% RSLogix 500 project 07_P10_ASHLEY_J.RSS, saved by version 8.30.00.16 %
PROJECT "UNTITLED"    % processor: Bul.1763 MicroLogix 1100 Series B %

PROGRAM FILES
  LAD 2 "MAIN"  5 rungs
  LAD 3 "IO"  8 rungs
  LAD 4 "HOA_CTRLS"  10 rungs
  LAD 5 "CONTROLS"  7 rungs
  LAD 6 "ALARMS"  14 rungs

DATA FILES
  O0 OUTPUT  4 elements
  I1 INPUT  6 elements
  S2 STATUS  66 elements
  B3 BINARY  10 elements
  T4 TIMER  4 elements
  C5 COUNTER  1 elements
  R6 CONTROL  1 elements
  N7 INTEGER  4 elements
  F8 FLOAT  1 elements

LADDER 2 "MAIN"
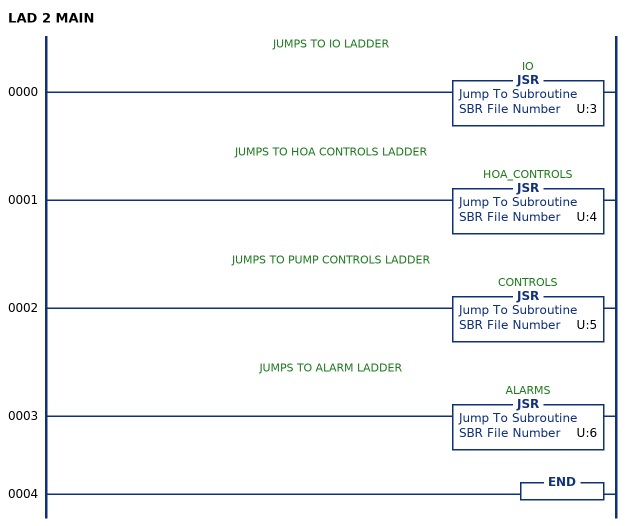
% Rung: 0 %
% JUMPS TO IO LADDER %
SOR JSR U:3 EOR
%   U:3  "IO" %
% Rung: 1 %
% JUMPS TO HOA CONTROLS LADDER %
SOR JSR U:4 EOR
%   U:4  "HOA_CONTROLS" %
% Rung: 2 %
% JUMPS TO PUMP CONTROLS LADDER %
SOR JSR U:5 EOR
%   U:5  "CONTROLS" %
% Rung: 3 %
% JUMPS TO ALARM LADDER %
SOR JSR U:6 EOR
%   U:6  "ALARMS" %
% Rung: 4 %
SOR END EOR

LADDER 3 "IO"
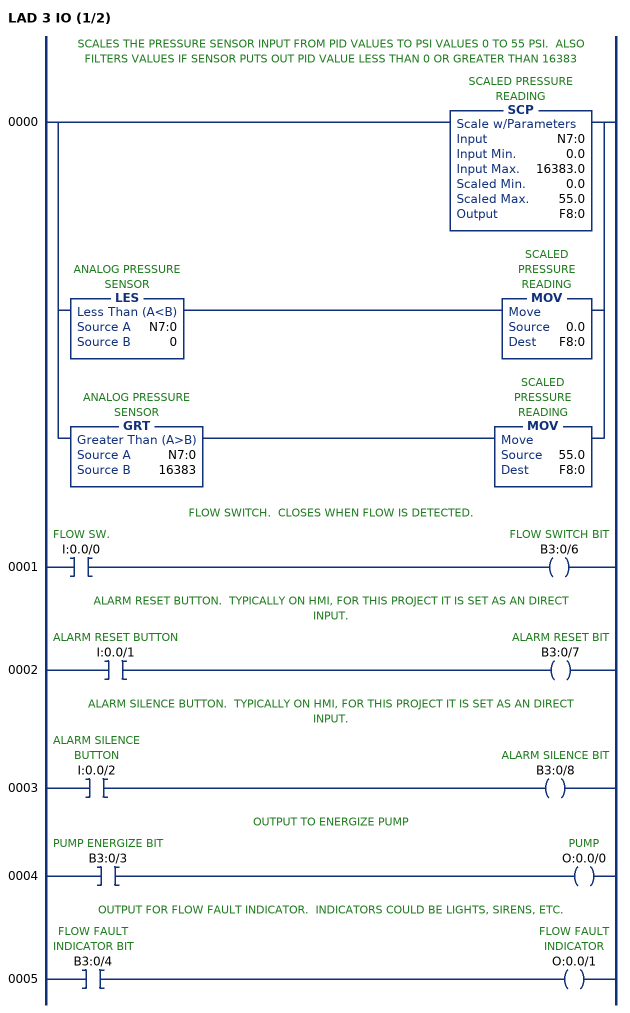
% Rung: 0 %
% SCALES THE PRESSURE SENSOR INPUT FROM PID VALUES TO PSI VALUES 0 TO 55 PSI.  ALSO FILTERS VALUES IF SENSOR PUTS OUT PID VALUE LESS THAN 0 OR GREATER THAN 16383 %
SOR BST SCP N7:0 0.0 16383.0 0.0 55.0 F8:0 NXB LES N7:0 0 MOV 0.0 F8:0 NXB GRT N7:0 16383 MOV 55.0 F8:0 BND EOR
%   N7:0  "ANALOG PRESSURE SENSOR" %
%   F8:0  "SCALED PRESSURE READING" %
% Rung: 1 %
% FLOW SWITCH.  CLOSES WHEN FLOW IS DETECTED. %
SOR XIC I:0.0/0 OTE B3:0/6 EOR
%   I:0.0/0  "FLOW SW." %
%   B3:0/6  "FLOW SWITCH BIT" %
% Rung: 2 %
% ALARM RESET BUTTON.  TYPICALLY ON HMI, FOR THIS PROJECT IT IS SET AS AN DIRECT INPUT. %
SOR XIC I:0.0/1 OTE B3:0/7 EOR
%   I:0.0/1  "ALARM RESET BUTTON" %
%   B3:0/7  "ALARM RESET BIT" %
% Rung: 3 %
% ALARM SILENCE BUTTON.  TYPICALLY ON HMI, FOR THIS PROJECT IT IS SET AS AN DIRECT INPUT. %
SOR XIC I:0.0/2 OTE B3:0/8 EOR
%   I:0.0/2  "ALARM SILENCE BUTTON" %
%   B3:0/8  "ALARM SILENCE BIT" %
% Rung: 4 %
% OUTPUT TO ENERGIZE PUMP %
SOR XIC B3:0/3 OTE O:0.0/0 EOR
%   B3:0/3  "PUMP ENERGIZE BIT" %
%   O:0.0/0  "PUMP" %
% Rung: 5 %
% OUTPUT FOR FLOW FAULT INDICATOR.  INDICATORS COULD BE LIGHTS, SIRENS, ETC. %
SOR XIC B3:0/4 OTE O:0.0/1 EOR
%   B3:0/4  "FLOW FAULT INDICATOR BIT" %
%   O:0.0/1  "FLOW FAULT INDICATOR" %

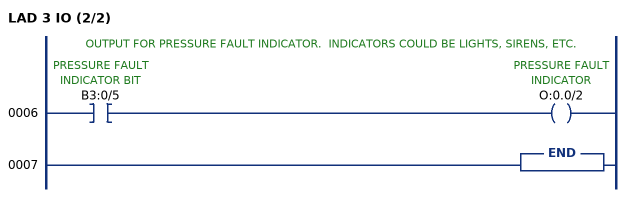
% Rung: 6 %
% OUTPUT FOR PRESSURE FAULT INDICATOR.  INDICATORS COULD BE LIGHTS, SIRENS, ETC. %
SOR XIC B3:0/5 OTE O:0.0/2 EOR
%   B3:0/5  "PRESSURE FAULT INDICATOR BIT" %
%   O:0.0/2  "PRESSURE FAULT INDICATOR" %
% Rung: 7 %
SOR END EOR

LADDER 4 "HOA_CTRLS"
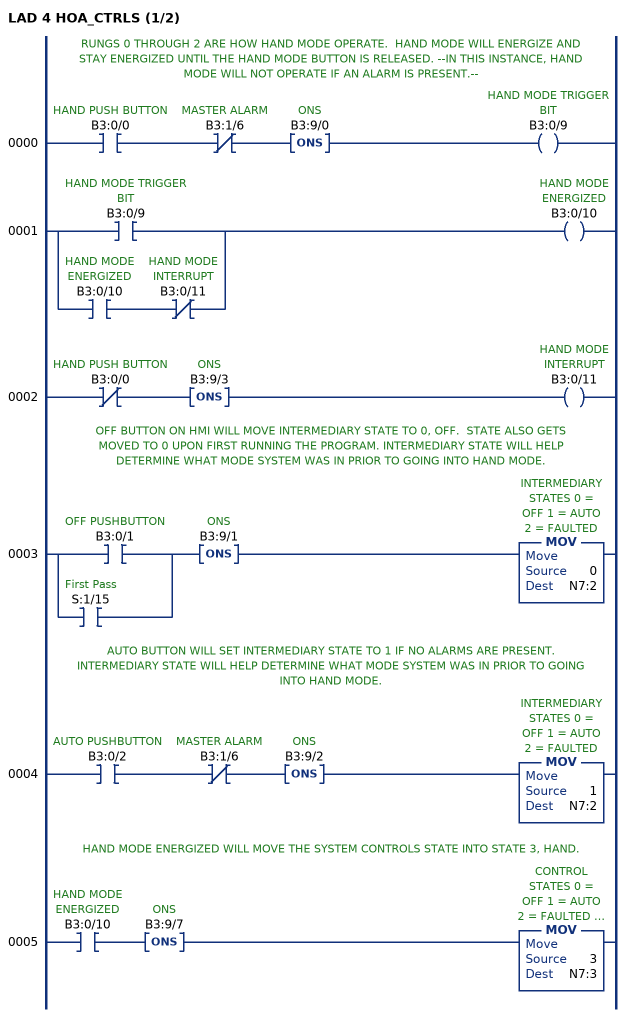
% Rung: 0 %
% RUNGS 0 THROUGH 2 ARE HOW HAND MODE OPERATE.  HAND MODE WILL ENERGIZE AND STAY ENERGIZED UNTIL THE HAND MODE BUTTON IS RELEASED. --IN THIS INSTANCE, HAND MODE WILL NOT OPERATE IF AN ALARM IS PRESENT.-- %
SOR XIC B3:0/0 XIO B3:1/6 ONS B3:9/0 OTE B3:0/9 EOR
%   B3:0/0  "HAND PUSH BUTTON" %
%   B3:1/6  "MASTER ALARM" %
%   B3:9/0  "ONS" %
%   B3:0/9  "HAND MODE TRIGGER BIT" %
% Rung: 1 %
SOR BST XIC B3:0/9 NXB XIC B3:0/10 XIO B3:0/11 BND OTE B3:0/10 EOR
%   B3:0/9  "HAND MODE TRIGGER BIT" %
%   B3:0/10  "HAND MODE ENERGIZED" %
%   B3:0/11  "HAND MODE INTERRUPT" %
% Rung: 2 %
SOR XIO B3:0/0 ONS B3:9/3 OTE B3:0/11 EOR
%   B3:0/0  "HAND PUSH BUTTON" %
%   B3:9/3  "ONS" %
%   B3:0/11  "HAND MODE INTERRUPT" %
% Rung: 3 %
% OFF BUTTON ON HMI WILL MOVE INTERMEDIARY STATE TO 0, OFF.  STATE ALSO GETS MOVED TO 0 UPON FIRST RUNNING THE PROGRAM. INTERMEDIARY STATE WILL HELP DETERMINE WHAT MODE SYSTEM WAS IN PRIOR TO GOING INTO HAND MODE. %
SOR BST XIC B3:0/1 NXB XIC S:1/15 BND ONS B3:9/1 MOV 0 N7:2 EOR
%   B3:0/1  "OFF PUSHBUTTON" %
%   S:1/15  "First Pass" %
%   B3:9/1  "ONS" %
%   N7:2  "INTERMEDIARY STATES 0 = OFF 1 = AUTO 2 = FAULTED" %
% Rung: 4 %
% AUTO BUTTON WILL SET INTERMEDIARY STATE TO 1 IF NO ALARMS ARE PRESENT.  INTERMEDIARY STATE WILL HELP DETERMINE WHAT MODE SYSTEM WAS IN PRIOR TO GOING INTO HAND MODE. %
SOR XIC B3:0/2 XIO B3:1/6 ONS B3:9/2 MOV 1 N7:2 EOR
%   B3:0/2  "AUTO PUSHBUTTON" %
%   B3:1/6  "MASTER ALARM" %
%   B3:9/2  "ONS" %
%   N7:2  "INTERMEDIARY STATES 0 = OFF 1 = AUTO 2 = FAULTED" %
% Rung: 5 %
% HAND MODE ENERGIZED WILL MOVE THE SYSTEM CONTROLS STATE INTO STATE 3, HAND. %
SOR XIC B3:0/10 ONS B3:9/7 MOV 3 N7:3 EOR
%   B3:0/10  "HAND MODE ENERGIZED" %
%   B3:9/7  "ONS" %
%   N7:3  "CONTROL STATES 0 = OFF 1 = AUTO 2 = FAULTED 3 = HAND" %

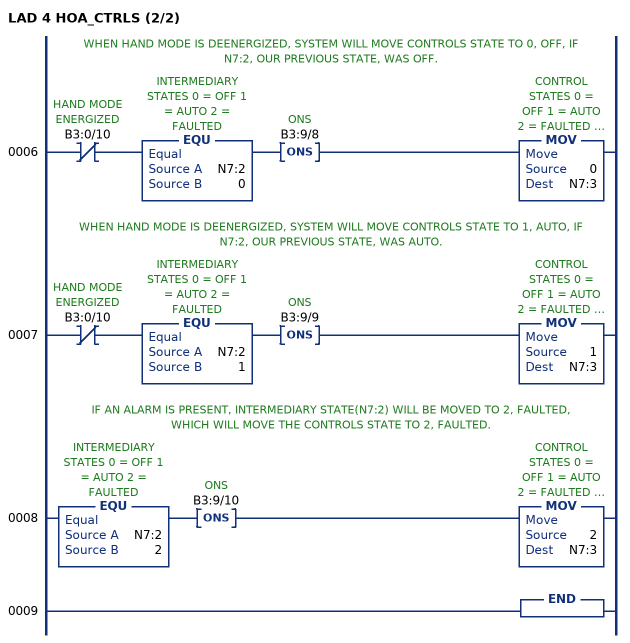
% Rung: 6 %
% WHEN HAND MODE IS DEENERGIZED, SYSTEM WILL MOVE CONTROLS STATE TO 0, OFF, IF N7:2, OUR PREVIOUS STATE, WAS OFF. %
SOR XIO B3:0/10 EQU N7:2 0 ONS B3:9/8 MOV 0 N7:3 EOR
%   B3:0/10  "HAND MODE ENERGIZED" %
%   N7:2  "INTERMEDIARY STATES 0 = OFF 1 = AUTO 2 = FAULTED" %
%   B3:9/8  "ONS" %
%   N7:3  "CONTROL STATES 0 = OFF 1 = AUTO 2 = FAULTED 3 = HAND" %
% Rung: 7 %
% WHEN HAND MODE IS DEENERGIZED, SYSTEM WILL MOVE CONTROLS STATE TO 1, AUTO, IF N7:2, OUR PREVIOUS STATE, WAS AUTO. %
SOR XIO B3:0/10 EQU N7:2 1 ONS B3:9/9 MOV 1 N7:3 EOR
%   B3:0/10  "HAND MODE ENERGIZED" %
%   N7:2  "INTERMEDIARY STATES 0 = OFF 1 = AUTO 2 = FAULTED" %
%   B3:9/9  "ONS" %
%   N7:3  "CONTROL STATES 0 = OFF 1 = AUTO 2 = FAULTED 3 = HAND" %
% Rung: 8 %
% IF AN ALARM IS PRESENT, INTERMEDIARY STATE(N7:2) WILL BE MOVED TO 2, FAULTED, WHICH WILL MOVE THE CONTROLS STATE TO 2, FAULTED. %
SOR EQU N7:2 2 ONS B3:9/10 MOV 2 N7:3 EOR
%   N7:2  "INTERMEDIARY STATES 0 = OFF 1 = AUTO 2 = FAULTED" %
%   B3:9/10  "ONS" %
%   N7:3  "CONTROL STATES 0 = OFF 1 = AUTO 2 = FAULTED 3 = HAND" %
% Rung: 9 %
SOR END EOR

LADDER 5 "CONTROLS"
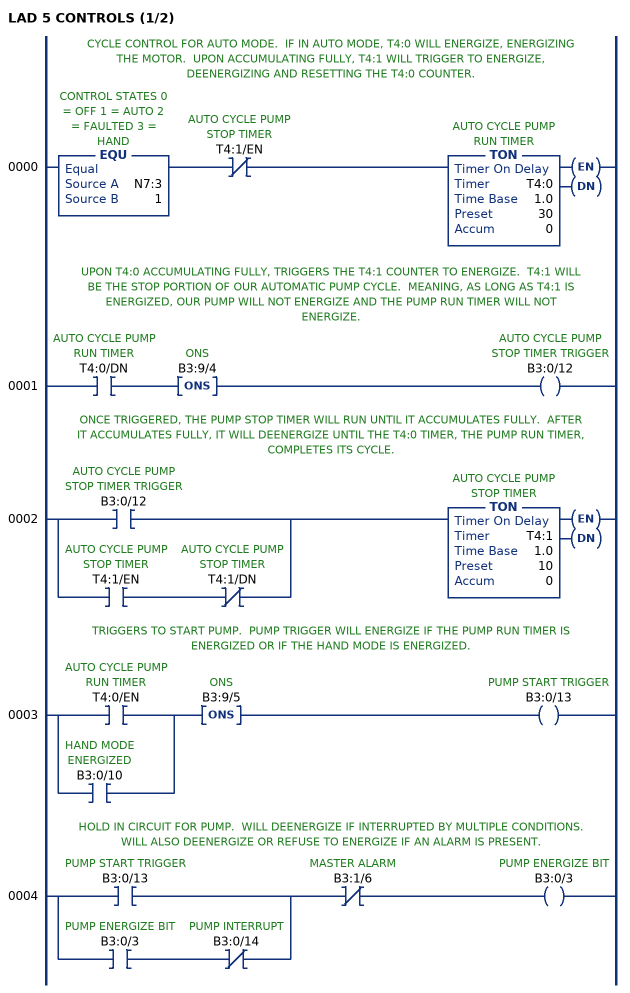
% Rung: 0 %
% CYCLE CONTROL FOR AUTO MODE.  IF IN AUTO MODE, T4:0 WILL ENERGIZE, ENERGIZING THE MOTOR.  UPON ACCUMULATING FULLY, T4:1 WILL TRIGGER TO ENERGIZE, DEENERGIZING AND RESETTING THE T4:0 COUNTER. %
SOR EQU N7:3 1 XIO T4:1/EN TON T4:0 1.0 30 0 EOR
%   N7:3  "CONTROL STATES 0 = OFF 1 = AUTO 2 = FAULTED 3 = HAND" %
%   T4:1  "AUTO CYCLE PUMP STOP TIMER" %
%   T4:0  "AUTO CYCLE PUMP RUN TIMER" %
% Rung: 1 %
% UPON T4:0 ACCUMULATING FULLY, TRIGGERS THE T4:1 COUNTER TO ENERGIZE.  T4:1 WILL BE THE STOP PORTION OF OUR AUTOMATIC PUMP CYCLE.  MEANING, AS LONG AS T4:1 IS ENERGIZED, OUR PUMP WILL NOT ENERGIZE AND THE PUMP RUN TIMER WILL NOT ENERGIZE. %
SOR XIC T4:0/DN ONS B3:9/4 OTE B3:0/12 EOR
%   T4:0  "AUTO CYCLE PUMP RUN TIMER" %
%   B3:9/4  "ONS" %
%   B3:0/12  "AUTO CYCLE PUMP STOP TIMER TRIGGER" %
% Rung: 2 %
% ONCE TRIGGERED, THE PUMP STOP TIMER WILL RUN UNTIL IT ACCUMULATES FULLY.  AFTER IT ACCUMULATES FULLY, IT WILL DEENERGIZE UNTIL THE T4:0 TIMER, THE PUMP RUN TIMER, COMPLETES ITS CYCLE. %
SOR BST XIC B3:0/12 NXB XIC T4:1/EN XIO T4:1/DN BND TON T4:1 1.0 10 0 EOR
%   B3:0/12  "AUTO CYCLE PUMP STOP TIMER TRIGGER" %
%   T4:1  "AUTO CYCLE PUMP STOP TIMER" %
% Rung: 3 %
% TRIGGERS TO START PUMP.  PUMP TRIGGER WILL ENERGIZE IF THE PUMP RUN TIMER IS ENERGIZED OR IF THE HAND MODE IS ENERGIZED. %
SOR BST XIC T4:0/EN NXB XIC B3:0/10 BND ONS B3:9/5 OTE B3:0/13 EOR
%   T4:0  "AUTO CYCLE PUMP RUN TIMER" %
%   B3:0/10  "HAND MODE ENERGIZED" %
%   B3:9/5  "ONS" %
%   B3:0/13  "PUMP START TRIGGER" %
% Rung: 4 %
% HOLD IN CIRCUIT FOR PUMP.  WILL DEENERGIZE IF INTERRUPTED BY MULTIPLE CONDITIONS.  WILL ALSO DEENERGIZE OR REFUSE TO ENERGIZE IF AN ALARM IS PRESENT. %
SOR BST XIC B3:0/13 NXB XIC B3:0/3 XIO B3:0/14 BND XIO B3:1/6 OTE B3:0/3 EOR
%   B3:0/13  "PUMP START TRIGGER" %
%   B3:0/3  "PUMP ENERGIZE BIT" %
%   B3:0/14  "PUMP INTERRUPT" %
%   B3:1/6  "MASTER ALARM" %

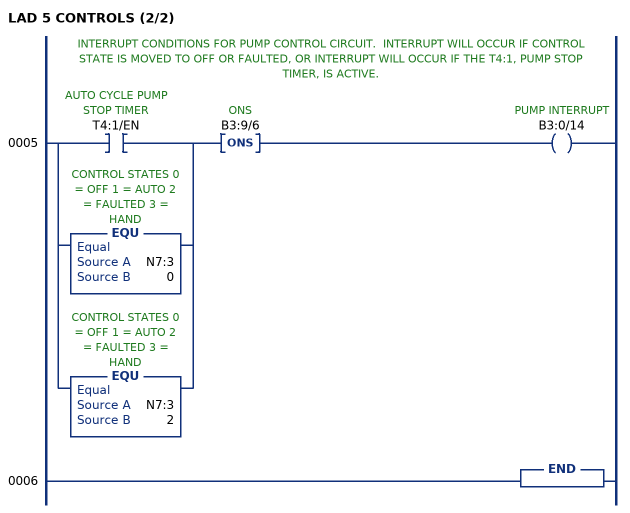
% Rung: 5 %
% INTERRUPT CONDITIONS FOR PUMP CONTROL CIRCUIT.  INTERRUPT WILL OCCUR IF CONTROL STATE IS MOVED TO OFF OR FAULTED, OR INTERRUPT WILL OCCUR IF THE T4:1, PUMP STOP TIMER, IS ACTIVE. %
SOR BST XIC T4:1/EN NXB EQU N7:3 0 NXB EQU N7:3 2 BND ONS B3:9/6 OTE B3:0/14 EOR
%   T4:1  "AUTO CYCLE PUMP STOP TIMER" %
%   N7:3  "CONTROL STATES 0 = OFF 1 = AUTO 2 = FAULTED 3 = HAND" %
%   B3:9/6  "ONS" %
%   B3:0/14  "PUMP INTERRUPT" %
% Rung: 6 %
SOR END EOR

LADDER 6 "ALARMS"
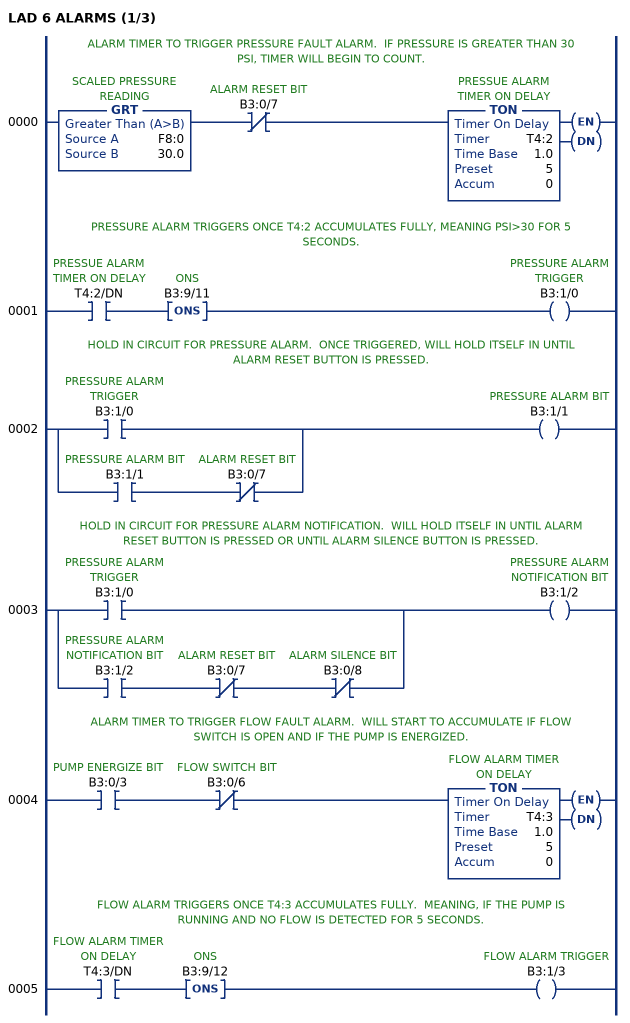
% Rung: 0 %
% ALARM TIMER TO TRIGGER PRESSURE FAULT ALARM.  IF PRESSURE IS GREATER THAN 30 PSI, TIMER WILL BEGIN TO COUNT. %
SOR GRT F8:0 30.0 XIO B3:0/7 TON T4:2 1.0 5 0 EOR
%   F8:0  "SCALED PRESSURE READING" %
%   B3:0/7  "ALARM RESET BIT" %
%   T4:2  "PRESSUE ALARM TIMER ON DELAY" %
% Rung: 1 %
% PRESSURE ALARM TRIGGERS ONCE T4:2 ACCUMULATES FULLY, MEANING PSI>30 FOR 5 SECONDS. %
SOR XIC T4:2/DN ONS B3:9/11 OTE B3:1/0 EOR
%   T4:2  "PRESSUE ALARM TIMER ON DELAY" %
%   B3:9/11  "ONS" %
%   B3:1/0  "PRESSURE ALARM TRIGGER" %
% Rung: 2 %
% HOLD IN CIRCUIT FOR PRESSURE ALARM.  ONCE TRIGGERED, WILL HOLD ITSELF IN UNTIL ALARM RESET BUTTON IS PRESSED. %
SOR BST XIC B3:1/0 NXB XIC B3:1/1 XIO B3:0/7 BND OTE B3:1/1 EOR
%   B3:1/0  "PRESSURE ALARM TRIGGER" %
%   B3:1/1  "PRESSURE ALARM BIT" %
%   B3:0/7  "ALARM RESET BIT" %
% Rung: 3 %
% HOLD IN CIRCUIT FOR PRESSURE ALARM NOTIFICATION.  WILL HOLD ITSELF IN UNTIL ALARM RESET BUTTON IS PRESSED OR UNTIL ALARM SILENCE BUTTON IS PRESSED. %
SOR BST XIC B3:1/0 NXB XIC B3:1/2 XIO B3:0/7 XIO B3:0/8 BND OTE B3:1/2 EOR
%   B3:1/0  "PRESSURE ALARM TRIGGER" %
%   B3:1/2  "PRESSURE ALARM NOTIFICATION BIT" %
%   B3:0/7  "ALARM RESET BIT" %
%   B3:0/8  "ALARM SILENCE BIT" %
% Rung: 4 %
% ALARM TIMER TO TRIGGER FLOW FAULT ALARM.  WILL START TO ACCUMULATE IF FLOW SWITCH IS OPEN AND IF THE PUMP IS ENERGIZED. %
SOR XIC B3:0/3 XIO B3:0/6 TON T4:3 1.0 5 0 EOR
%   B3:0/3  "PUMP ENERGIZE BIT" %
%   B3:0/6  "FLOW SWITCH BIT" %
%   T4:3  "FLOW ALARM TIMER ON DELAY" %
% Rung: 5 %
% FLOW ALARM TRIGGERS ONCE T4:3 ACCUMULATES FULLY.  MEANING, IF THE PUMP IS RUNNING AND NO FLOW IS DETECTED FOR 5 SECONDS. %
SOR XIC T4:3/DN ONS B3:9/12 OTE B3:1/3 EOR
%   T4:3  "FLOW ALARM TIMER ON DELAY" %
%   B3:9/12  "ONS" %
%   B3:1/3  "FLOW ALARM TRIGGER" %

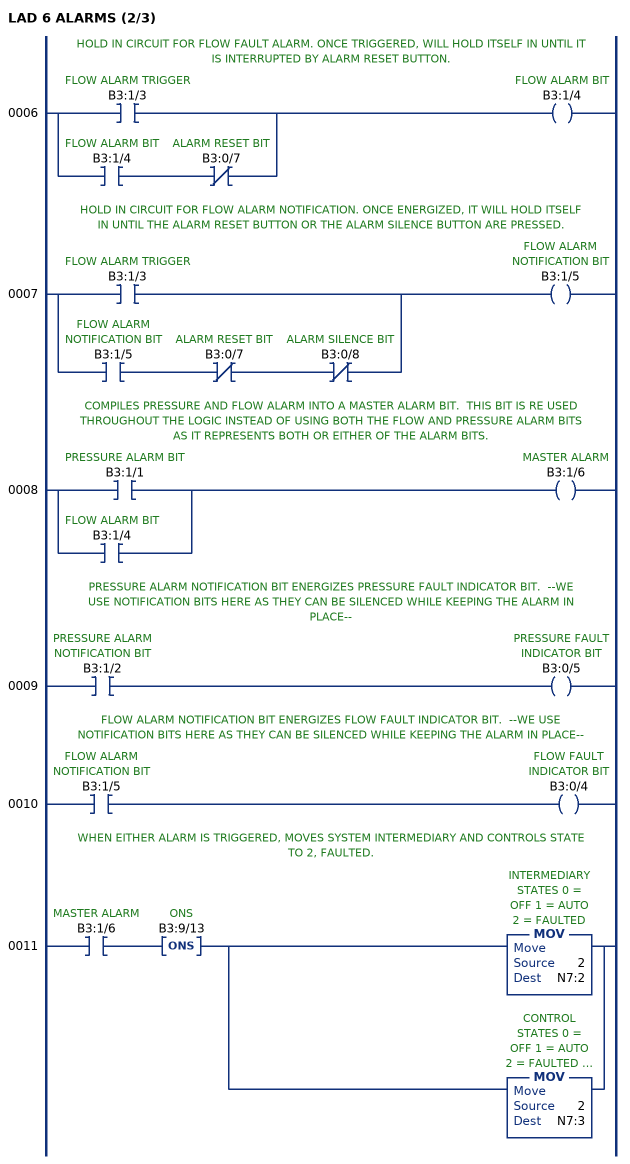
% Rung: 6 %
% HOLD IN CIRCUIT FOR FLOW FAULT ALARM. ONCE TRIGGERED, WILL HOLD ITSELF IN UNTIL IT IS INTERRUPTED BY ALARM RESET BUTTON. %
SOR BST XIC B3:1/3 NXB XIC B3:1/4 XIO B3:0/7 BND OTE B3:1/4 EOR
%   B3:1/3  "FLOW ALARM TRIGGER" %
%   B3:1/4  "FLOW ALARM BIT" %
%   B3:0/7  "ALARM RESET BIT" %
% Rung: 7 %
% HOLD IN CIRCUIT FOR FLOW ALARM NOTIFICATION. ONCE ENERGIZED, IT WILL HOLD ITSELF IN UNTIL THE ALARM RESET BUTTON OR THE ALARM SILENCE BUTTON ARE PRESSED. %
SOR BST XIC B3:1/3 NXB XIC B3:1/5 XIO B3:0/7 XIO B3:0/8 BND OTE B3:1/5 EOR
%   B3:1/3  "FLOW ALARM TRIGGER" %
%   B3:1/5  "FLOW ALARM NOTIFICATION BIT" %
%   B3:0/7  "ALARM RESET BIT" %
%   B3:0/8  "ALARM SILENCE BIT" %
% Rung: 8 %
% COMPILES PRESSURE AND FLOW ALARM INTO A MASTER ALARM BIT.  THIS BIT IS RE USED THROUGHOUT THE LOGIC INSTEAD OF USING BOTH THE FLOW AND PRESSURE ALARM BITS AS IT REPRESENTS BOTH OR EITHER OF THE ALARM BITS. %
SOR BST XIC B3:1/1 NXB XIC B3:1/4 BND OTE B3:1/6 EOR
%   B3:1/1  "PRESSURE ALARM BIT" %
%   B3:1/4  "FLOW ALARM BIT" %
%   B3:1/6  "MASTER ALARM" %
% Rung: 9 %
% PRESSURE ALARM NOTIFICATION BIT ENERGIZES PRESSURE FAULT INDICATOR BIT.  --WE USE NOTIFICATION BITS HERE AS THEY CAN BE SILENCED WHILE KEEPING THE ALARM IN PLACE-- %
SOR XIC B3:1/2 OTE B3:0/5 EOR
%   B3:1/2  "PRESSURE ALARM NOTIFICATION BIT" %
%   B3:0/5  "PRESSURE FAULT INDICATOR BIT" %
% Rung: 10 %
% FLOW ALARM NOTIFICATION BIT ENERGIZES FLOW FAULT INDICATOR BIT.  --WE USE NOTIFICATION BITS HERE AS THEY CAN BE SILENCED WHILE KEEPING THE ALARM IN PLACE-- %
SOR XIC B3:1/5 OTE B3:0/4 EOR
%   B3:1/5  "FLOW ALARM NOTIFICATION BIT" %
%   B3:0/4  "FLOW FAULT INDICATOR BIT" %
% Rung: 11 %
% WHEN EITHER ALARM IS TRIGGERED, MOVES SYSTEM INTERMEDIARY AND CONTROLS STATE TO 2, FAULTED. %
SOR XIC B3:1/6 ONS B3:9/13 BST MOV 2 N7:2 NXB MOV 2 N7:3 BND EOR
%   B3:1/6  "MASTER ALARM" %
%   B3:9/13  "ONS" %
%   N7:2  "INTERMEDIARY STATES 0 = OFF 1 = AUTO 2 = FAULTED" %
%   N7:3  "CONTROL STATES 0 = OFF 1 = AUTO 2 = FAULTED 3 = HAND" %

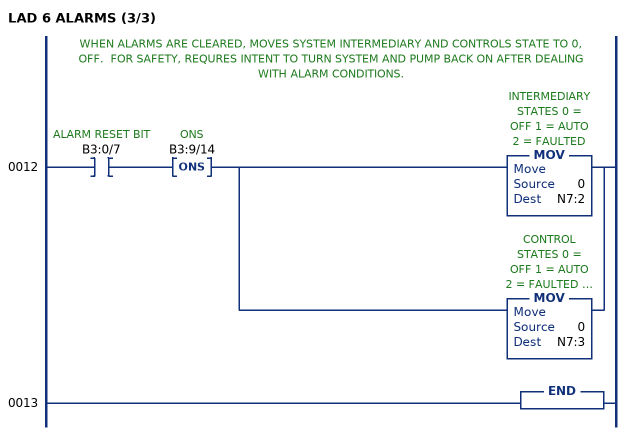
% Rung: 12 %
% WHEN ALARMS ARE CLEARED, MOVES SYSTEM INTERMEDIARY AND CONTROLS STATE TO 0, OFF.  FOR SAFETY, REQURES INTENT TO TURN SYSTEM AND PUMP BACK ON AFTER DEALING WITH ALARM CONDITIONS. %
SOR XIC B3:0/7 ONS B3:9/14 BST MOV 0 N7:2 NXB MOV 0 N7:3 BND EOR
%   B3:0/7  "ALARM RESET BIT" %
%   B3:9/14  "ONS" %
%   N7:2  "INTERMEDIARY STATES 0 = OFF 1 = AUTO 2 = FAULTED" %
%   N7:3  "CONTROL STATES 0 = OFF 1 = AUTO 2 = FAULTED 3 = HAND" %
% Rung: 13 %
SOR END EOR

OTHER DOCUMENTED ADDRESSES
  B3:0/15  "AUTO CYCLE PUMP START TRIGGER"
  B3:9/15  "ONS"

DATA TABLE (non-zero values as saved)
DATA T4
% .PRE .ACC %
% T4:0 % 30 0
% T4:1 % 10 0
% T4:2 % 5 0
% T4:3 % 5 0
